PROGRAM MAIN
VAR
    fbMotionLogger : FB_MotionLogger; // Shared resource
    // Persistant storage
    fbPersistentDataStorage : FB_PersistentDataStorage; // Shared resource
    M1 : ST_MotionEpicsItf; // shared ressource

	{attribute 'pytmc':='pv: TST:SmartAct:MCS2-3C'}
    {attribute 'TcLinkTo' := '
		.fbEncoderScaling.nRawEncoderDINT :=TIID^Master_EtherCAT^MCS2-3C^Module 1 (MCS2M-D-3C)^mode/status/pos/fError TxPDO^Position Actual Value;
        .fbMotionAxis.stDS402Drive.stDriveStatus	:=TIID^Master_EtherCAT^MCS2-3C^Module 1 (MCS2M-D-3C)^mode/status/pos/fError TxPDO^Status Word;
        .fbMotionAxis.stDS402Drive.nFollowingError		:=TIID^Master_EtherCAT^MCS2-3C^Module 1 (MCS2M-D-3C)^mode/status/pos/fError TxPDO^Following Error Actual Value;
        .fbMotionAxis.stDS402Drive.nModeOfOperation		:=TIID^Master_EtherCAT^MCS2-3C^Module 1 (MCS2M-D-3C)^ctl/mode/pos/vel/acc RxPDO^Modes of Operation;     
		.fbMotionAxis.stDS402Drive.nModeOfOperationDisplay:=TIID^Master_EtherCAT^MCS2-3C^Module 1 (MCS2M-D-3C)^mode/status/pos/fError TxPDO^Modes of Operation Display;
		.fbMotionAxis.stDS402Drive.nDS402DriveControl	:=TIID^Master_EtherCAT^MCS2-3C^Module 1 (MCS2M-D-3C)^ctl/mode/pos/vel/acc RxPDO^Control Word;
    '}
   {attribute 'TcLinkToOSO' := '
        .fbMotionAxis.stDS402Drive.nModeOfOperationNC	:=<0,8,0>TINC^NC-Task 1 SAF^Axes^MCS2-M1^Drive^Outputs^Out^nCtrl5;   
        .fbMotionAxis.stDS402Drive.nDS402DriveControlNC := <0,8,0>TINC^NC-Task 1 SAF^Axes^MCS2-M1^Drive^Outputs^Out^nCtrl1;
        .fbMotionAxis.stDS402Drive.nDS402DriveControlNC := <8,8,0>TINC^NC-Task 1 SAF^Axes^MCS2-M1^Drive^Outputs^Out^nCtrl2;
    '}
    fbMotionStage : FB_MotionStageMCS2(	sName := 'MCS2',
                                        stMotionEpicsItf := M1,
                                        AxisRef := NcAxis_GVL.MCS2,
                                        iMotionLogger := fbMotionLogger,
                                        iPersistentDataStorage := fbPersistentDataStorage
                                    ) := (BrakeMode := E_StageBrakeMode.IF_MOVING, EnableMode:=ENUM_StageEnableMode.DURING_MOTION, HomeMode:=E_EpicsHomeCmd.AUTOZERO);
    
    bHardEnable AT %Q*: BOOL := TRUE;
END_VAR

fbMotionLogger();
fbPersistentDataStorage();
fbMotionStage();

END_PROGRAM

(* stored: Version 1.1.0.1
   POU MAIN: Id {61c6dfbc-a7dc-4c03-9ea3-aa217d748554}, SpecialFunc None *)
